//{attribute 'qualified_only'}
VAR_GLOBAL
	bWaterSensor 			AT %I*	: BOOL;
	diWaterverbruikVandaag			: DINT;
END_VAR

(* stored: Version 1.1.0.1
   GVL GVL_Energiemetingen: Id {2f302f60-f326-4f2a-b06b-35329b1b8ed2} *)
